// TIA Portal V17 export
// export: Created 2025-03-05T08:02:18.1389483Z, ExportSetting WithDefaults, DisplayName Totally Integrated Automation Portal, DisplayVersion V17 Update 8, DisplayName TIA Portal Openness, DisplayVersion V17 Update 8, DisplayName TIA Portal Version Control Interface, DisplayVersion V17, DisplayName SINAMICS Startdrive Advanced, DisplayVersion V17 SP2, DisplayName SINAMICS Startdrive G110M, G120, G120C, G120D, G120P, G115D, DisplayVersion V17 SP2, DisplayName SINAMICS Startdrive G130, G150, S120, S150, SINAMICS MV, S210, DisplayVersion V17 SP2, DisplayName STEP 7 Professional, DisplayVersion V17 Update 8, DisplayName SINUMERIK ONE STEP 7 Toolbox, DisplayVersion V17 Update 12, DisplayName SINUMERIK 840D sl STEP 7 Toolbox, DisplayVersion V17 Update 12, DisplayName STEP 7 Safety, DisplayVersion V17 Update 6, DisplayName WinCC Advanced, DisplayVersion V17 Update 8
TYPE "HT10_OUTPUTS"
// stored: IsFailsafeCompliant false
   STRUCT
      SPARE_0_0 : Bool;   // SPARE 0 0
      RESET_FAULT_Q : Bool;   // HT10 RESET FAULT OUTPUT
      SPARE_1 : Byte;   // SPARE 1
      SPARE_2_0 : Bool;   // SPARE 2 0
      SPARE_2_1 : Bool;   // SPARE 2 1
      SPARE_2_2 : Bool;   // SPARE 2 2
      SPARE_2_3 : Bool;   // SPARE 2 3
      SPARE_2_4 : Bool;   // SPARE 2 4
      SPARE_2_5 : Bool;   // SPARE 2 5
      SPARE_2_6 : Bool;   // SPARE 2 6
      JOG_PLUS_Q : Bool;   // HT10 JOG PLUS OUTPUT
      SPARE_3_0 : Bool;   // SPARE 3 0
      SPARE_3_1 : Bool;   // SPARE 3 1
      SPARE_3_2 : Bool;   // SPARE 3 2
      SPARE_3_3 : Bool;   // SPARE 3 3
      SPARE_3_4 : Bool;   // SPARE 3 4
      SPARE_3_5 : Bool;   // SPARE 3 5
      JOG_MIINUS_Q : Bool;   // HT10 JOG MIINUS OUTPUT
      SPARE_3_7 : Bool;   // SPARE 3 7
      SPARE_4 : Byte;   // SPARE 4
      RAPID_Q : Bool;   // HT10 RAPID OUTPUT
      SPARE_5_1 : Bool;   // SPARE 5 1
      SPARE_5_2 : Bool;   // SPARE 5 2
      SPARE_5_3 : Bool;   // SPARE 5 3
      SPARE_5_4 : Bool;   // SPARE 5 4
      SPARE_5_5 : Bool;   // SPARE 5 5
      SPARE_5_6 : Bool;   // SPARE 5 6
      SPARE_5_7 : Bool;   // SPARE 5 7
      NC_STOP_Q : Bool;   // HT10 NC STOP OUTPUT
      NC_START_Q : Bool;   // HT10 NC START OUTPUT
   END_STRUCT;
END_TYPE
